FUNCTION DisposeNode : BOOL
VAR_INPUT
	node : I_Node;
END_VAR
VAR
	disposableNode : I_Disposable;
END_VAR

IF __QUERYINTERFACE(node,disposableNode) THEN
 	disposableNode.Dispose();
	DisposeNode := TRUE;
END_IF;

END_FUNCTION

(* stored: Version 1.1.0.1, ProductVersion 3.1.4024.12
   POU DisposeNode: Id {c412776f-3e2d-0642-38f7-75ac19500c35}, SpecialFunc None *)
